fbSP_TemperatureLow(
	xEnable:= TRUE,		//rTemperature > 0,			//Temperature can drop below 0C
	rInput:= rTemperature, 
	rSwitchPoint:= rThresholdTemperatureLow_int, 
	rHysteresis:= 3, 
	xInvert:= TRUE, 
	xOut=> );
fbEI_TemperatureLow.sInstanceName := sInstanceName;
fbEI_TemperatureLow.sErrorInfo := TO_STRING(_Domoticz_RoundDecimals(rTemperature,1));
fbEI_TemperatureLow.sErrorInfo := CONCAT(fbEI_TemperatureLow.sErrorInfo, ' C');
fbEI_TemperatureLow(
	scConnector:= scConnector,
	xError:= fbSP_TemperatureLow.xOut
			AND rThresholdTemperatureLow_int > 0
			AND uiIdentifier_TempHumBaro > 0,
	eErrorID:= Domoticz_eErrors.Tasmota_TemperatureLow
);

//********************************************HUMIDITY
fbSP_HumidityHigh(	
	xEnable:= rHumidity > 0,								//If humidity not used (Temp or TempBaro)
	rInput:= rHumidity, 
	rSwitchPoint:= rThresholdHumidityHigh_int, 
	rHysteresis:= 10, 
	xInvert:= FALSE, 
	xOut=> );
fbEI_HumidityHigh.sInstanceName := sInstanceName;
fbEI_HumidityHigh.sErrorInfo := TO_STRING(TO_INT(_Domoticz_RoundDecimals(rHumidity,0)));
fbEI_HumidityHigh.sErrorInfo := CONCAT(fbEI_HumidityHigh.sErrorInfo, ' %');
fbEI_HumidityHigh(
	scConnector:= scConnector,
	xError:= fbSP_HumidityHigh.xOut 
			AND rThresholdHumidityHigh_int > 0
			AND uiIdentifier_TempHumBaro > 0,
	eErrorID:= Domoticz_eErrors.Tasmota_HumidityHigh
);

fbSP_HumidityLow(
	xEnable:= rHumidity > 0,								//If humidity not used (Temp or TempBaro)
	rInput:= rHumidity, 
	rSwitchPoint:= rThresholdHumidityLow_int, 
	rHysteresis:= 10, 
	xInvert:= TRUE, 
	xOut=> );
fbEI_HumidityLow.sInstanceName := sInstanceName;
fbEI_HumidityLow.sErrorInfo := TO_STRING(TO_INT(_Domoticz_RoundDecimals(rHumidity,0)));
fbEI_HumidityLow.sErrorInfo := CONCAT(fbEI_HumidityLow.sErrorInfo, ' %');
fbEI_HumidityLow(
	scConnector:= scConnector,
	xError:= fbSP_HumidityLow.xOut 							
			AND rThresholdHumidityLow_int > 0
			AND uiIdentifier_TempHumBaro > 0,
	eErrorID:= Domoticz_eErrors.Tasmota_HumidityLow
);

//********************************************CARBON DIOXIDE
fbSP_CarbonDioxideHigh(
	xEnable:= rCarbonDioxide > 0,
	rInput:= rCarbonDioxide, 
	rSwitchPoint:= rThresholdCarbonDioxideHigh_int, 
	rHysteresis:= 250, 
	xInvert:= FALSE, 
	xOut=> );
fbEI_CarbonDioxideHigh.sInstanceName := sInstanceName;
fbEI_CarbonDioxideHigh.sErrorInfo := TO_STRING(TO_INT(_Domoticz_RoundDecimals(rCarbonDioxide,0)));
fbEI_CarbonDioxideHigh.sErrorInfo := CONCAT(fbEI_CarbonDioxideHigh.sErrorInfo, ' ppm');
fbEI_CarbonDioxideHigh(
	scConnector:= scConnector,
	xError:= fbSP_CarbonDioxideHigh.xOut 
			AND rThresholdCarbonDioxideHigh_int > 0
			AND uiIdentifier_CarbonDioxide > 0,
	eErrorID:= Domoticz_eErrors.Tasmota_CarbondioxideHigh
);

fbSP_CarbonDioxideCritical(
	xEnable:= rCarbonDioxide > 0,
	rInput:= rCarbonDioxide, 
	rSwitchPoint:= rThresholdCarbonDioxideCritical_int, 
	rHysteresis:= 250, 
	xInvert:= FALSE, 
	xOut=> );
fbEI_CarbonDioxideCritical.sInstanceName := sInstanceName;
fbEI_CarbonDioxideCritical.sErrorInfo := TO_STRING(TO_INT(_Domoticz_RoundDecimals(rCarbonDioxide,0)));
fbEI_CarbonDioxideCritical.sErrorInfo := CONCAT(fbEI_CarbonDioxideCritical.sErrorInfo, ' ppm');
fbEI_CarbonDioxideCritical(
	scConnector:= scConnector,
	xError:= fbSP_CarbonDioxideCritical.xOut 
			AND rThresholdCarbonDioxideCritical_int > 0
			AND uiIdentifier_CarbonDioxide > 0,
	eErrorID:= Domoticz_eErrors.Tasmota_CarbonDioxideCritical
);

//********************************************PARTICLES
fbSP_1umHigh(
	xEnable:= rParticles_1um > 0,
	rInput:= rParticles_1um, 
	rSwitchPoint:= rThresholdParticlesHigh_1um_int, 
	rHysteresis:= 10, 
	xInvert:= FALSE, 
	xOut=> );
fbEI_1umHigh.sInstanceName := sInstanceName;
fbEI_1umHigh.sErrorInfo := TO_STRING(_Domoticz_RoundDecimals(rParticles_1um,1));
fbEI_1umHigh.sErrorInfo := CONCAT(fbEI_1umHigh.sErrorInfo, ' ug/m3');
fbEI_1umHigh(
	scConnector:= scConnector,
	xError:= fbSP_1umHigh.xOut
			AND rThresholdParticlesHigh_1um_int > 0
			AND uiIdentifier_1um > 0,
	eErrorID:= Domoticz_eErrors.Tasmota_ParticlesHigh_1um
);

fbSP_2_5umHigh(
	xEnable:= rParticles_2_5um > 0,
	rInput:= rParticles_2_5um, 
	rSwitchPoint:= rThresholdParticlesHigh_2_5um_int, 
	rHysteresis:= 10, 
	xInvert:= FALSE, 
	xOut=> );
fbEI_2_5umHigh.sInstanceName := sInstanceName;
fbEI_2_5umHigh.sErrorInfo := TO_STRING(_Domoticz_RoundDecimals(rParticles_2_5um,1));
fbEI_2_5umHigh.sErrorInfo := CONCAT(fbEI_2_5umHigh.sErrorInfo, ' ug/m3');
fbEI_2_5umHigh(
	scConnector:= scConnector,
	xError:= fbSP_2_5umHigh.xOut 
			AND rThresholdParticlesHigh_2_5um_int > 0
			AND uiIdentifier_2_5um > 0,
	eErrorID:= Domoticz_eErrors.Tasmota_ParticlesHigh_2_5um
);

fbSP_10umHigh(	
	xEnable:= rParticles_10um > 0,
	rInput:= rParticles_10um,
	rSwitchPoint:= rThresholdParticlesHigh_10um_int, 
	rHysteresis:= 10, 
	xInvert:= FALSE, 
	xOut=> );
fbEI_10umHigh.sInstanceName := sInstanceName;
fbEI_10umHigh.sErrorInfo := TO_STRING(_Domoticz_RoundDecimals(rParticles_10um,1));
fbEI_10umHigh.sErrorInfo := CONCAT(fbEI_10umHigh.sErrorInfo, ' ug/m3');
fbEI_10umHigh(
	scConnector:= scConnector,
	xError:= fbSP_10umHigh.xOut 
			AND rThresholdParticlesHigh_10um_int > 0
			AND uiIdentifier_10um > 0,
	eErrorID:= Domoticz_eErrors.Tasmota_ParticlesHigh_10um
);
END_ACTION

{attribute 'monitoring' := 'call'} PROPERTY rThresholdCurrentHigh :REAL
SET
rThresholdCurrentHigh_int := rThresholdCurrentHigh;
END_SET
GET
rThresholdCurrentHigh := rThresholdCurrentHigh_int;
END_GET
END_PROPERTY

{attribute 'monitoring' := 'call'} PROPERTY rThresholdCurrentMax :REAL
SET
rThresholdCurrentMax_int := rThresholdCurrentMax;
END_SET
GET
rThresholdCurrentMax := rThresholdCurrentMax_int;
END_GET
END_PROPERTY

{attribute 'monitoring' := 'call'} PROPERTY rThresholdPowerUsageHigh :REAL
SET
rThresholdPowerUsageHigh_int := rThresholdPowerUsageHigh;
END_SET
GET
rThresholdPowerUsageHigh := rThresholdPowerUsageHigh_int;
END_GET
END_PROPERTY

{attribute 'monitoring' := 'call'} PROPERTY rThresholdPowerUsageToday :REAL
SET
rThresholdPowerUsageToday_int := rThresholdPowerUsageToday;
END_SET
GET
rThresholdPowerUsageToday := rThresholdPowerUsageToday_int;
END_GET
END_PROPERTY

{attribute 'monitoring' := 'call'} PROPERTY rThresholdTemperatureHigh :REAL
SET
rThresholdTemperatureHigh_int := rThresholdTemperatureHigh;
END_SET
GET
rThresholdTemperatureHigh := rThresholdTemperatureHigh_int;
END_GET
END_PROPERTY

{attribute 'monitoring' := 'call'} PROPERTY rThresholdTemperatureLow :REAL
SET
rThresholdTemperatureLow_int := rThresholdTemperatureLow;
END_SET
GET
rThresholdTemperatureLow := rThresholdTemperatureLow_int;
END_GET
END_PROPERTY

{attribute 'monitoring' := 'call'} PROPERTY rThresholdHumidityHigh :REAL
SET
rThresholdHumidityHigh_int := rThresholdHumidityHigh;
END_SET
GET
rThresholdHumidityHigh := rThresholdHumidityHigh_int;
END_GET
END_PROPERTY

{attribute 'monitoring' := 'call'} PROPERTY rThresholdHumidityLow :REAL
SET
rThresholdHumidityLow_int := rThresholdHumidityLow;
END_SET
GET
rThresholdHumidityLow := rThresholdHumidityLow_int;
END_GET
END_PROPERTY

{attribute 'monitoring' := 'call'} PROPERTY rThresholdCarbonDioxideHigh :REAL
SET
rThresholdCarbonDioxideHigh_int := rThresholdCarbonDioxideHigh;
END_SET
GET
rThresholdCarbonDioxideHigh := rThresholdCarbonDioxideHigh_int;
END_GET
END_PROPERTY

{attribute 'monitoring' := 'call'} PROPERTY rThresholdCarbonDioxideCritical :REAL
SET
rThresholdCarbonDioxideCritical_int := rThresholdCarbonDioxideCritical;
END_SET
GET
rThresholdCarbonDioxideCritical := rThresholdCarbonDioxideCritical_int;
END_GET
END_PROPERTY

{attribute 'monitoring' := 'call'} PROPERTY rThresholdParticlesHigh_1um :REAL
SET
rThresholdParticlesHigh_1um_int := rThresholdParticlesHigh_1um;
END_SET
GET
rThresholdParticlesHigh_1um := rThresholdParticlesHigh_1um_int;
END_GET
END_PROPERTY

{attribute 'monitoring' := 'call'} PROPERTY rThresholdParticlesHigh_2_5um :REAL
SET
rThresholdParticlesHigh_2_5um_int := rThresholdParticlesHigh_2_5um;
END_SET
GET
rThresholdParticlesHigh_2_5um := rThresholdParticlesHigh_2_5um_int;
END_GET
END_PROPERTY

{attribute 'monitoring' := 'call'} PROPERTY rThresholdParticlesHigh_10um :REAL
SET
rThresholdParticlesHigh_10um_int := rThresholdParticlesHigh_10um;
END_SET
GET
rThresholdParticlesHigh_10um := rThresholdParticlesHigh_10um_int;
END_GET
END_PROPERTY

PROPERTY rThresholdVoltage : REAL
SET
rThresholdVoltage_int := rThresholdVoltage;
END_SET
GET
rThresholdVoltage := rThresholdVoltage_int;
END_GET
END_PROPERTY

END_FUNCTION_BLOCK

// Function Blocks/Hardware/Devices/Domoticz_GoogleDevices
{attribute 'conditionalshow_all_locals'}
FUNCTION_BLOCK Domoticz_GoogleDevices EXTENDS _Domoticz_Connector_InOut	//Don't use xForceValues for everything because it will also force byMediaControl_Set
VAR_INPUT
	uiIdentifier_Status			:UINT;	//Device Status
	uiIdentifier_Source			:UINT;	//Source of active footage
	uiIdentifier_Volume			:UINT;	//Device Volume
	byVolume_Set				:BYTE;	//Volume (0-100)
	uiIdentifier_MediaControl	:UINT;	//Process Usage
	byMediaControl_Set			:BYTE;	//Play process (0-100)
	xMediaControl_Set			:BOOL;	//Play media
END_VAR
VAR_OUTPUT
	sStatus						:STRING(Domoticz_Constants.uiMaxSValuesize);
	bySource					:BYTE;	//See domoticz settings! Default:0=off, 10=Spotify, 20=Netflix, 30=Youtube, 40=Other
	byVolume_Act				:BYTE;
	byMediaControl_Act			:BYTE;
	xMediaControl_Act			:BOOL;
END_VAR
VAR
	afb_ObjectString_Out		:ARRAY[1..1] OF _Domoticz_ObjectString_Out;
	afb_ObjectInt_Out			:ARRAY[1..1] OF _Domoticz_ObjectInt_Out;
	afb_ObjectInt_InOut			:ARRAY[1..2] OF _Domoticz_ObjectInt_InOut;
	afb_ObjectBool_InOut		:ARRAY[1..1] OF _Domoticz_ObjectBool_InOut;
END_VAR

IF __ISVALIDREF(scConnector) THEN
	Main();
END_IF

ACTION Main:
{attribute 'conditionalshow'}
//Call parent function
SUPER^.Main();

//Call all 
afb_ObjectString_Out[1].tDataTimeOut := T#24H;
afb_ObjectString_Out[1](scConnector := scConnector,		uiIdentifier := uiIdentifier_Status,		rxUpdateInterlock := rxUpdateInterlock_int,			sValueAct => sStatus);

afb_ObjectInt_Out[1].tDataTimeOut := T#24H;
afb_ObjectInt_Out[1](	scConnector := scConnector,		uiIdentifier := uiIdentifier_Source,		rxUpdateInterlock := rxUpdateInterlock_int);

afb_ObjectInt_InOut[1].tDataTimeOut := T#24H;
afb_ObjectInt_InOut[1].iValueSetLimitLow := -1;
afb_ObjectInt_InOut[1].iValueSetLimitHigh := 101;
afb_ObjectInt_InOut[1].eCommandType := _Domoticz_eCommandType.SetBrightness;
afb_ObjectInt_InOut[1](	scConnector := scConnector, 	uiIdentifier := uiIdentifier_Volume,		rxUpdateInterlock := rxUpdateInterlock_int,			iValueSet := byVolume_Set);

afb_ObjectInt_InOut[2].tDataTimeOut := T#24H;
afb_ObjectInt_InOut[2].iValueSetLimitLow := -1;
afb_ObjectInt_InOut[2].iValueSetLimitHigh := 101;
afb_ObjectInt_InOut[2].eCommandType := _Domoticz_eCommandType.SetBrightness;
afb_ObjectInt_InOut[2](	scConnector := scConnector, 	uiIdentifier := uiIdentifier_MediaControl,	rxUpdateInterlock := rxUpdateInterlock_int,			iValueSet := byMediaControl_Set);

afb_ObjectBool_InOut[1].tDataTimeOut := T#24H;      
afb_ObjectBool_InOut[1].eCommandType := _Domoticz_eCommandType.SwitchLight;                                                 
afb_ObjectBool_InOut[1](scConnector := scConnector,		uiIdentifier := uiIdentifier_MediaControl,	rxUpdateInterlock := rxUpdateInterlock_int,			xValueSet := xMediaControl_Set,		xValueAct => xMediaControl_Act);
						
//Output
bySource 			:= TO_BYTE(afb_ObjectInt_Out[1].iValueAct);
byVolume_Act 		:= TO_BYTE(afb_ObjectInt_InOut[1].iValueAct);
byMediaControl_Act 	:= TO_BYTE(afb_ObjectInt_InOut[2].iValueAct);
 
//Force update of volume
IF xForceSetValues AND byVolume_Set <> byVolume_Act THEN
	afb_ObjectInt_InOut[1].ForceSet(tForceSetValues_int);
END_IF

//Force update of media control
IF xForceSetValues AND byMediaControl_Set <> byMediaControl_Act THEN
	afb_ObjectInt_InOut[2].ForceSet(tForceSetValues_int);
END_IF

//Force update of media control
IF xForceSetValues AND xMediaControl_Set <> xMediaControl_Act THEN
	afb_ObjectBool_InOut[1].ForceSet(tForceSetValues_int);
END_IF
										   
//Errors
fbEI_DataTimeOut.sInstanceName := sInstanceName;
fbEI_DataTimeOut.tErrorDelay := T#500MS;	//Give objects time to be overruled by other updates
fbEI_DataTimeOut(
	scConnector:= scConnector,
	xError:= xDataTimeOut_int
			AND (afb_ObjectString_Out[1].xDataTimedOut
			OR afb_ObjectInt_Out[1].xDataTimedOut
			OR afb_ObjectInt_InOut[1].xDataTimedOut
			OR afb_ObjectInt_InOut[2].xDataTimedOut
			OR afb_ObjectBool_InOut[1].xDataTimedOut),
	eErrorID:= Domoticz_eErrors.ObjectDataTimeOut
);
END_ACTION

END_FUNCTION_BLOCK

// Function Blocks/Hardware/Custom/Domoticz_CustomString
{attribute 'conditionalshow_all_locals'}
FUNCTION_BLOCK Domoticz_CustomString EXTENDS _Domoticz_Connector_InOut_Extended
VAR_INPUT
	uiIdentifier				:UINT;	//Device to control
	sValueSet					:STRING(Domoticz_Constants.uiMaxSValuesize);
END_VAR
VAR_OUTPUT
	sValueAct					:STRING(Domoticz_Constants.uiMaxSValuesize);
END_VAR
VAR
	afb_ObjectString_InOut		:ARRAY[1..1] OF _Domoticz_ObjectString_InOut;
END_VAR

IF __ISVALIDREF(scConnector) THEN
	Main();
END_IF

ACTION Main:
{attribute 'conditionalshow'}
//Call parent function
SUPER^.Main();

//Call all functions
afb_ObjectString_InOut[1].tDataTimeOut := tDataTimeOut_int;
afb_ObjectString_InOut[1](scConnector := scConnector, 	uiIdentifier := uiIdentifier,	sValueSet := sValueSet, 	sValueAct => sValueAct);

//Force status if enabled
IF xForceSetValues AND sValueSet <> sValueAct THEN
	afb_ObjectString_InOut[1].ForceSet(tForceSetValues_int);
END_IF

//Errors
fbEI_DataTimeOut.sInstanceName := sInstanceName;
fbEI_DataTimeOut.tErrorDelay := T#500MS;	//Give objects TIME TO be overruled BY other updates
fbEI_DataTimeOut(
	scConnector:= scConnector,
	xError:= xDataTimeOut_int
			AND (afb_ObjectString_InOut[1].xDataTimedOut),
	eErrorID:= Domoticz_eErrors.ObjectDataTimeOut
);
END_ACTION

END_FUNCTION_BLOCK

// Function Blocks/Hardware/Climate/Energy/Domoticz_UsageMeter
{attribute 'conditionalshow_all_locals'}
FUNCTION_BLOCK Domoticz_UsageMeter EXTENDS _Domoticz_Connector_Out
VAR_INPUT
	uiIdentifier_Usage			:UINT;			//Usage (cumulative)
	xPulse						:BOOL;			//Measure pulse
	rUnitsPerPulse				:REAL := 1000;	//Units per pulse
	rUnitsBeforeUpdate			:REAL := 1000;	//Amount of units to reach before sending update
	tTimeOutPulse				:TIME := T#5M;	//Time to pass without pulses to sens stored values
END_VAR                          
VAR_OUTPUT                       
	rUsageToday					:REAL;
	rUsageCumulative			:REAL;
END_VAR                          
VAR	                             
	afb_ObjectArrayReal_InOut	:ARRAY[1..1] OF _Domoticz_ObjectArrayReal_InOut;
	xPulse_old					:BOOL;
	TON_TimeOutPulse			:TON;
	                             
	rThresholdUsageToday_int	:REAL := 500;
	fbEI_UsageToday				:Domoticz_ErrorInterface;
	
	sUnit_int					:STRING := 'm3';
END_VAR                          
VAR PERSISTENT RETAIN                 
	rPulsesCounted				:REAL;
END_VAR

IF __ISVALIDREF(scConnector) THEN
	Main();
END_IF

ACTION Main:
{attribute 'conditionalshow'}
//Call parent function
SUPER^.Main();

//Add usage on pulse
IF xPulse AND NOT xPulse_old THEN
	xPulse_old := TRUE;
	//Add pulses if limit not reached, set data to zero
	IF ((rPulsesCounted+1)*rUnitsPerPulse) < rUnitsBeforeUpdate THEN
		rPulsesCounted := rPulsesCounted + 1;
		afb_ObjectArrayReal_InOut[1].arValueSet[Domoticz_eSValues_Usage.Usage] := 0;
	//Limit reached, send data and reset counter
	ELSIF ((rPulsesCounted+1)*rUnitsPerPulse) >= rUnitsBeforeUpdate THEN
		afb_ObjectArrayReal_InOut[1].arValueSet[Domoticz_eSValues_Usage.Usage] := rUnitsBeforeUpdate;
		rPulsesCounted := 0;
	END_IF
//Reset flank
ELSIF NOT xPulse THEN
	xPulse_old := FALSE;
END_IF
	
//Send usage after timeout to prevent values buildup
IF TON_TimeOutPulse.Q THEN
	afb_ObjectArrayReal_InOut[1].arValueSet[Domoticz_eSValues_Usage.Usage] := rPulsesCounted*rUnitsPerPulse;
	rPulsesCounted := 0;
END_IF

//Call all functions
afb_ObjectArrayReal_InOut[1].tDataTimeOut := T#15M;
afb_ObjectArrayReal_InOut[1].eDataSource := _Domoticz_eDataSource.HTTP;
afb_ObjectArrayReal_InOut[1](scConnector := scConnector, 	uiIdentifier := uiIdentifier_Usage);

//Call timer
TON_TimeOutPulse(IN:= NOT xPulse, PT:= tTimeOutPulse);

//Outputs
rUsageToday := afb_ObjectArrayReal_InOut[1].arValueAct[Domoticz_eSValues_Usage.UsageToday];
rUsageCumulative := afb_ObjectArrayReal_InOut[1].arValueAct[Domoticz_eSValues_Usage.UsageCumulative];

//Errors
//********************************************DATA
fbEI_DataTimeOut.sInstanceName := sInstanceName;
fbEI_DataTimeOut.tErrorDelay := T#500MS;	//Give objects TIME TO be overruled BY other updates
fbEI_DataTimeOut(
	scConnector:= scConnector,
	xError:= xDataTimeOut_int
			AND (afb_ObjectArrayReal_InOut[1].xDataTimedOut),
	eErrorID:= Domoticz_eErrors.ObjectDataTimeOut
);

//********************************************USAGE TODAY
fbEI_UsageToday.sInstanceName := sInstanceName;
fbEI_UsageToday.sErrorInfo := TO_STRING(_Domoticz_RoundDecimals(rUsageToday,2));
fbEI_UsageToday.sErrorInfo := CONCAT(fbEI_UsageToday.sErrorInfo, ' ');
fbEI_UsageToday.sErrorInfo := CONCAT(fbEI_UsageToday.sErrorInfo, sUnit_int);
fbEI_UsageToday(
	scConnector:= scConnector,
	xError:= (rUsageToday > rThresholdUsageToday_int) 
			AND rThresholdUsageToday_int > 0
			AND uiIdentifier_Usage > 0,
	eErrorID:= Domoticz_eErrors.UsageMeter_UsageToday
);
END_ACTION

{attribute 'monitoring' := 'call'} PROPERTY rThresholdUsageToday :REAL
SET
rThresholdUsageToday_int := rThresholdUsageToday;
END_SET
GET
rThresholdUsageToday := rThresholdUsageToday_int;
END_GET
END_PROPERTY

PROPERTY sUnit : STRING
SET
sUnit_int := sUnit;
END_SET
GET
sUnit := sUnit_int;
END_GET
END_PROPERTY

END_FUNCTION_BLOCK

// Function Blocks/Hardware/Devices/Domoticz_Life360
{attribute 'conditionalshow_all_locals'}
//Function block to update sentire values in domoticz
FUNCTION_BLOCK Domoticz_Life360 EXTENDS _Domoticz_Connector_Out
VAR_INPUT
	uiIdentifier_Presence				:UINT;	//Presence at home
	uiIdentifier_Location				:UINT;	//Current location (text)
	uiIdentifier_Battery				:UINT;	//Device battery (%)
	uiIdentifier_Distance				:UINT;	//Distance to home
END_VAR
VAR_OUTPUT
	xPresence							:BOOL;
	sLocation							:STRING;
	rBattery							:REAL;
	sDistance							:STRING;
END_VAR
VAR
	afb_ObjectReal_Out					:ARRAY[1..1] OF _Domoticz_ObjectReal_Out;
	afb_ObjectString_Out				:ARRAY[1..2] OF _Domoticz_ObjectString_Out;		
	afb_ObjectBool_Out					:ARRAY[1..1] OF _Domoticz_ObjectBool_Out;
	
	xArrivedHome_int					:BOOL := TRUE;
	fbEI_ArrivedHome					:Domoticz_ErrorInterface;
	
	xLeftHome_int						:BOOL := TRUE;
	fbEI_LeftHome						:Domoticz_ErrorInterface;
	
END_VAR

IF __ISVALIDREF(scConnector) THEN
	Main();
END_IF

ACTION Main:
{attribute 'conditionalshow'}
//Call parent function
SUPER^.Main();

//Call all functions
//Data timeout assume normal workweek - excluding weekends
afb_ObjectReal_Out[1].tDataTimeOut := T#3D;
afb_ObjectReal_Out[1](scConnector := scConnector, 	uiIdentifier := uiIdentifier_Battery,		rxUpdateInterlock := rxUpdateInterlock_int,			rValueAct => rBattery);
                                                                                            	                                                	
afb_ObjectBool_Out[1].tDataTimeOut := T#3D;                                                 	                                                	
afb_ObjectBool_Out[1](scConnector:= scConnector, 	uiIdentifier:= uiIdentifier_Presence,		rxUpdateInterlock := rxUpdateInterlock_int,			xValueAct => xPresence);
                                                                                            	                                                	
afb_ObjectString_Out[1].tDataTimeOut := T#3D;                                               	                                                	
afb_ObjectString_Out[1](scConnector := scConnector,	uiIdentifier := uiIdentifier_Location,		rxUpdateInterlock := rxUpdateInterlock_int,			sValueAct => sLocation);
                                                                                            	                                                	
afb_ObjectString_Out[2].tDataTimeOut := T#3D;                                               	                                                	
afb_ObjectString_Out[2](scConnector := scConnector,	uiIdentifier := uiIdentifier_Distance, 		rxUpdateInterlock := rxUpdateInterlock_int,			sValueAct => sDistance);

//Errors
fbEI_DataTimeOut.sInstanceName := sInstanceName;
fbEI_DataTimeOut.tErrorDelay := T#500MS;	//Give objects TIME TO be overruled BY other updates
fbEI_DataTimeOut(
	scConnector:= scConnector,
	xError:= xDataTimeOut_int
			AND (afb_ObjectReal_Out[1].xDataTimedOut
			OR afb_ObjectBool_Out[1].xDataTimedOut
			OR afb_ObjectString_Out[1].xDataTimedOut
			OR afb_ObjectString_Out[2].xDataTimedOut),
	eErrorID:= Domoticz_eErrors.ObjectDataTimeOut
);

fbEI_ArrivedHome.sInstanceName := sInstanceName;
fbEI_ArrivedHome(
	scConnector:= scConnector, 
	xError:= xPresence
			AND xArrivedHome_int, 
	eErrorID:= Domoticz_eErrors.Life360_ArrivedHome
);

fbEI_LeftHome.sInstanceName := sInstanceName;
fbEI_LeftHome(
	scConnector:= scConnector, 
	xError:= NOT xPresence
			AND xleftHome_int, 
	eErrorID:= Domoticz_eErrors.Life360_LeftHome
);
END_ACTION

PROPERTY xArrivedHome :BOOL
SET
xArrivedHome_int := xArrivedHome;
END_SET
GET
xArrivedHome := xArrivedHome_int;
END_GET
END_PROPERTY

PROPERTY xLeftHome :BOOL
SET
xLeftHome_int := xLeftHome;
END_SET
GET
xLeftHome := xLeftHome_int;
END_GET
END_PROPERTY

END_FUNCTION_BLOCK

// Function Blocks/Hardware/Devices/Domoticz_HueSensor
{attribute 'conditionalshow_all_locals'}
//Function block to update sentire values in domoticz
FUNCTION_BLOCK Domoticz_HueSensor EXTENDS _Domoticz_Connector_Out
VAR_INPUT
	uiIdentifier_Temperature			:UINT;	//Temperature (C)
	uiIdentifier_Light					:UINT;	//Light level (lux)
	uiIdentifier_Ambient				:UINT;	//Ambient light level
	uiIdentifier_PIR					:UINT;	//PIR
END_VAR
VAR_OUTPUT
	rTemperature						:REAL;
	rLightIntensity						:REAL;
	xAmbient							:BOOL;
	xPIR								:BOOL;
END_VAR
VAR
	afb_ObjectReal_Out					:ARRAY[1..2] OF _Domoticz_ObjectReal_Out;
	afb_ObjectBool_Out					:ARRAY[1..2] OF _Domoticz_ObjectBool_Out;
END_VAR

IF __ISVALIDREF(scConnector) THEN
	Main();
END_IF

ACTION Main:
{attribute 'conditionalshow'}
//Call parent function
SUPER^.Main();

//Call all functions
//Data timeout Light/temp depend on amount of changes, assume 4h. Ambient switch at least twice a day
afb_ObjectReal_Out[1].tDataTimeOut := T#4H;
afb_ObjectReal_Out[1](scConnector:= scConnector,	uiIdentifier:= uiIdentifier_Temperature,		rxUpdateInterlock := rxUpdateInterlock_int,			rValueAct=> rTemperature);

afb_ObjectReal_Out[2].tDataTimeOut := T#8H;
afb_ObjectReal_Out[2](scConnector:= scConnector,	uiIdentifier:= uiIdentifier_Light,				rxUpdateInterlock := rxUpdateInterlock_int,			rValueAct=> rLightIntensity);

afb_ObjectBool_Out[1].tDataTimeOut := T#24H;	//Not guarded PIR
afb_ObjectBool_Out[1](scConnector:= scConnector, 	uiIdentifier:= uiIdentifier_PIR,				rxUpdateInterlock := rxUpdateInterlock_int,			xValueAct=> xPIR);

afb_ObjectBool_Out[2].tDataTimeOut := T#24H;
afb_ObjectBool_Out[2](scConnector:= scConnector, 	uiIdentifier:= uiIdentifier_Ambient,			rxUpdateInterlock := rxUpdateInterlock_int,			xValueAct=> xAmbient);									
										   
//Errors
fbEI_DataTimeOut.sInstanceName := sInstanceName;
fbEI_DataTimeOut.tErrorDelay := T#500MS;	//Give objects TIME TO be overruled BY other updates
fbEI_DataTimeOut(
	scConnector:= scConnector,
	xError:= xDataTimeOut_int
			AND (afb_ObjectReal_Out[1].xDataTimedOut
			OR afb_ObjectReal_Out[2].xDataTimedOut
			OR afb_ObjectBool_Out[1].xDataTimedOut
			OR afb_ObjectBool_Out[2].xDataTimedOut),
	eErrorID:= Domoticz_eErrors.ObjectDataTimeOut
);
END_ACTION

END_FUNCTION_BLOCK

// Function Blocks/Hardware/Devices/Domoticz_HuePlug
{attribute 'conditionalshow_all_locals'}
FUNCTION_BLOCK Domoticz_HuePlug EXTENDS _Domoticz_Connector_InOut
VAR_INPUT
	uiIdentifier				:UINT;	//Device to control
	xEnable						:BOOL;
END_VAR
VAR_OUTPUT
	xEnabled					:BOOL;
END_VAR
VAR
	afb_ObjectBool_InOut		:ARRAY[1..1] OF _Domoticz_ObjectBool_InOut;
END_VAR

IF __ISVALIDREF(scConnector) THEN
	Main();
END_IF

ACTION Main:
{attribute 'conditionalshow'}
//Call parent function
SUPER^.Main();

//Call all functions
afb_ObjectBool_InOut[1].tDataTimeOut := T#24H;
afb_ObjectBool_InOut[1].eCommandType := _Domoticz_eCommandType.SwitchLight;
afb_ObjectBool_InOut[1](scConnector := scConnector, 	uiIdentifier := uiIdentifier, 	xValueSet := xEnable, 	xValueAct => xEnabled);

//Force status if enabled
IF xForceSetValues AND xEnable <> xEnabled THEN
	afb_ObjectBool_InOut[1].ForceSet(tForceSetValues_int);
END_IF

//Errors
fbEI_DataTimeOut.sInstanceName := sInstanceName;
fbEI_DataTimeOut.tErrorDelay := T#500MS;	//Give objects TIME TO be overruled BY other updates
fbEI_DataTimeOut(
	scConnector:= scConnector,
	xError:= xDataTimeOut_int
			AND (afb_ObjectBool_InOut[1].xDataTimedOut),
	eErrorID:= Domoticz_eErrors.ObjectDataTimeOut
);
END_ACTION

END_FUNCTION_BLOCK

// Function Blocks/Hardware/Climate/Energy/Domoticz_P1Meter
{attribute 'conditionalshow_all_locals'}
FUNCTION_BLOCK Domoticz_P1Meter EXTENDS _Domoticz_Connector_Out
VAR_INPUT
	uiIdentifier_Voltage		:UINT;				//Usage
	uiIdentifier_Power			:UINT;				//Usage
	uiIdentifier_Gas			:UINT;				//Usage
	tUpdateRate					:TIME := T#60M;		//Used for data timeout
END_VAR                          
VAR_OUTPUT                       
	rVoltage					:REAL;
	rPowerUsageActual			:REAL;
	rPowerUsageToday			:REAL;
	rPowerUsageCumulative		:REAL;
	rPowerReturnActual			:REAL;
	rPowerReturnToday			:REAL;
	rPowerReturnCumulative		:REAL;
	rGasUsageToday				:REAL;
	rGasUsageCumulative			:REAL;
END_VAR                          
VAR	                             
	afb_ObjectReal_Out			:ARRAY[1..1] OF _Domoticz_ObjectReal_Out;
	afb_ObjectArrayReal_Out		:ARRAY[1..2] OF _Domoticz_ObjectArrayReal_Out;
	                             
	rThresholdVoltage_int		:REAL := 200;
	fbEI_PowerFailure			:Domoticz_ErrorInterface;
	                             
	rThresholdPowerUsageToday_int:REAL := 10.0; //kWh
	fbEI_PowerUsageToday		:Domoticz_ErrorInterface;
	                             
	rThresholdPowerUsageHigh_int:REAL := 3000;	//W
	fbSP_PowerUsageHigh			:_Domoticz_SwitchPoint;
	fbEI_PowerUsageHigh			:Domoticz_ErrorInterface;
	                             
	rThresholdGasUsageToday_int	:REAL := 5.0;	//m3
	fbEI_GasUsageToday			:Domoticz_ErrorInterface;
END_VAR

IF __ISVALIDREF(scConnector) THEN
	Main();
END_IF

ACTION Main:
{attribute 'conditionalshow'}
//Call parent function
SUPER^.Main();

//Call all functions
afb_ObjectReal_Out[1].tDataTimeOut := TO_TIME(TO_UDINT(tUpdateRate)*2);
afb_ObjectReal_Out[1](	scConnector := scConnector, 	uiIdentifier := uiIdentifier_Voltage, 		rxUpdateInterlock := rxUpdateInterlock_int,			rValueAct => rVoltage);

afb_ObjectArrayReal_Out[1].tDataTimeOut := TO_TIME(TO_UDINT(tUpdateRate)*2);
afb_ObjectArrayReal_Out[1](	scConnector := scConnector, uiIdentifier := uiIdentifier_Gas,			rxUpdateInterlock := rxUpdateInterlock_int);

afb_ObjectArrayReal_Out[2].tDataTimeOut := TO_TIME(TO_UDINT(tUpdateRate)*2);
afb_ObjectArrayReal_Out[2](scConnector := scConnector, 	uiIdentifier := uiIdentifier_Power,			rxUpdateInterlock := rxUpdateInterlock_int);

//Outputs
rGasUsageCumulative		:= afb_ObjectArrayReal_Out[1].arValueAct[Domoticz_eSValues_P1.Usage1Cumulative] + afb_ObjectArrayReal_Out[1].arValueAct[Domoticz_eSValues_P1.Usage2Cumulative];
rGasUsageToday			:= afb_ObjectArrayReal_Out[1].arValueAct[Domoticz_eSValues_P1.UsageToday];

rPowerUsageActual 		:= afb_ObjectArrayReal_Out[2].arValueAct[Domoticz_eSValues_P1.UsageActual];
rPowerReturnActual 		:= afb_ObjectArrayReal_Out[2].arValueAct[Domoticz_eSValues_P1.ReturnActual];
rPowerUsageCumulative 	:= afb_ObjectArrayReal_Out[2].arValueAct[Domoticz_eSValues_P1.Usage1Cumulative] + afb_ObjectArrayReal_Out[2].arValueAct[Domoticz_eSValues_P1.Usage2Cumulative];
rPowerReturnCumulative	:= afb_ObjectArrayReal_Out[2].arValueAct[Domoticz_eSValues_P1.Return1Cumulative] + afb_ObjectArrayReal_Out[2].arValueAct[Domoticz_eSValues_P1.Return2Cumulative];	
rPowerUsageToday 		:= afb_ObjectArrayReal_Out[2].arValueAct[Domoticz_eSValues_P1.UsageToday];
rPowerReturnToday 		:= afb_ObjectArrayReal_Out[2].arValueAct[Domoticz_eSValues_P1.ReturnToday];

//Errors
//********************************************DATA
fbEI_DataTimeOut.sInstanceName := sInstanceName;
fbEI_DataTimeOut.tErrorDelay := T#500MS;	//Give objects TIME TO be overruled BY other updates
fbEI_DataTimeOut(
	scConnector:= scConnector,
	xError:= xDataTimeOut_int
			AND (afb_ObjectReal_Out[1].xDataTimedOut
			OR afb_ObjectArrayReal_Out[1].xDataTimedOut
			OR afb_ObjectArrayReal_Out[2].xDataTimedOut),
	eErrorID:= Domoticz_eErrors.ObjectDataTimeOut
);

//********************************************POWER FAILURE
fbEI_PowerFailure.sInstanceName := sInstanceName;
fbEI_PowerFailure.sErrorInfo := TO_STRING(TO_INT(_Domoticz_RoundDecimals(rVoltage,0)));
fbEI_PowerFailure.sErrorInfo := CONCAT(fbEI_PowerFailure.sErrorInfo, ' V / ');
fbEI_PowerFailure.sErrorInfo := CONCAT(fbEI_PowerFailure.sErrorInfo, TO_STRING(TO_INT(_Domoticz_RoundDecimals(rPowerUsageActual,0))));
fbEI_PowerFailure.sErrorInfo := CONCAT(fbEI_PowerFailure.sErrorInfo, ' W');
fbEI_PowerFailure(
	scConnector:= scConnector,
	xError:= ((rVoltage < rThresholdVoltage_int) OR (rPowerUsageActual < 1)) 
			AND (uiIdentifier_Voltage > 0 OR  uiIdentifier_Power > 0),
	eErrorID:= Domoticz_eErrors.P1_PowerFailure
);

//********************************************USAGE TODAY
fbEI_PowerUsageToday.sInstanceName := sInstanceName;
fbEI_PowerUsageToday.sErrorInfo := TO_STRING(_Domoticz_RoundDecimals(rPowerUsageToday,2));
fbEI_PowerUsageToday.sErrorInfo := CONCAT(fbEI_PowerUsageToday.sErrorInfo, ' kWh');
fbEI_PowerUsageToday(
	scConnector:= scConnector,
	xError:= (rPowerUsageToday > rThresholdPowerUsageToday_int) 
			AND rThresholdPowerUsageToday_int > 0
			AND uiIdentifier_Power > 0,
	eErrorID:= Domoticz_eErrors.P1_PowerUsageToday
);

//********************************************USAGE
fbSP_PowerUsageHigh(
	xEnable:= rPowerUsageActual > 0,
	rInput:= rPowerUsageActual, 
	rSwitchPoint:= rThresholdPowerUsageHigh_int, 
	rHysteresis:= 500, 
	xInvert:= FALSE, 
	xOut=> );
fbEI_PowerUsageHigh.sInstanceName := sInstanceName;
fbEI_PowerUsageHigh.sErrorInfo := TO_STRING(TO_INT(_Domoticz_RoundDecimals(rPowerUsageActual,0)));
fbEI_PowerUsageHigh.sErrorInfo := CONCAT(fbEI_PowerUsageHigh.sErrorInfo, ' W');
fbEI_PowerUsageHigh(
	scConnector:= scConnector,
	xError:= fbSP_PowerUsageHigh.xOut
			AND rThresholdPowerUsageHigh_int > 0
			AND uiIdentifier_Power > 0,
	eErrorID:= Domoticz_eErrors.P1_PowerUsageHigh
);

//********************************************USAGE TODAY
fbEI_GasUsageToday.sInstanceName := sInstanceName;
fbEI_GasUsageToday.sErrorInfo := TO_STRING(_Domoticz_RoundDecimals(rGasUsageToday,2));
fbEI_GasUsageToday.sErrorInfo := CONCAT(fbEI_GasUsageToday.sErrorInfo, ' m3');
fbEI_GasUsageToday(
	scConnector:= scConnector,
	xError:= (rGasUsageToday > rThresholdGasUsageToday_int) 
			AND rThresholdGasUsageToday_int > 0
			AND uiIdentifier_Gas > 0,
	eErrorID:= Domoticz_eErrors.P1_GasUsageToday
);
END_ACTION

{attribute 'monitoring' := 'call'} PROPERTY rThresholdGasUsageToday :REAL
SET
rThresholdGasUsageToday_int := rThresholdGasUsageToday;
END_SET
GET
rThresholdGasUsageToday := rThresholdGasUsageToday_int;
END_GET
END_PROPERTY

{attribute 'monitoring' := 'call'} PROPERTY rThresholdPowerUsageHigh :REAL
SET
rThresholdPowerUsageHigh_int := rThresholdPowerUsageHigh;
END_SET
GET
rThresholdPowerUsageHigh := rThresholdPowerUsageHigh_int;
END_GET
END_PROPERTY

{attribute 'monitoring' := 'call'} PROPERTY rThresholdPowerUsageToday :REAL
SET
rThresholdPowerUsageToday_int := rThresholdPowerUsageToday;
END_SET
GET
rThresholdPowerUsageToday := rThresholdPowerUsageToday_int;
END_GET
END_PROPERTY

PROPERTY rThresholdVoltage : REAL
SET
rThresholdVoltage_int := rThresholdVoltage;
END_SET
GET
rThresholdVoltage := rThresholdVoltage_int;
END_GET
END_PROPERTY

END_FUNCTION_BLOCK

// Function Blocks/Hardware/Devices/Domoticz_HueSwitch
{attribute 'conditionalshow_all_locals'}
FUNCTION_BLOCK Domoticz_HueSwitch EXTENDS _Domoticz_Connector_Out
VAR_INPUT
	uiIdentifier				:UINT;	//Device to control
END_VAR
VAR_OUTPUT
	axButtons_Short				:ARRAY[1..4] OF BOOL;
	axButtons_Long				:ARRAY[1..4] OF BOOL;
END_VAR
VAR
	afb_ObjectInt_Out			:ARRAY[1..1] OF _Domoticz_ObjectInt_Out;
	wX							:WORD;
END_VAR

IF __ISVALIDREF(scConnector) THEN
	Main();
END_IF

ACTION Main:
{attribute 'conditionalshow'}
//Call parent function
SUPER^.Main();

//Call all functions
afb_ObjectInt_Out[1].tDataTimeOut := T#24H;
afb_ObjectInt_Out[1].eCommandType := _Domoticz_eCommandType.SwitchLight;
afb_ObjectInt_Out[1].eDataSource := _Domoticz_eDataSource.MQTT;
afb_ObjectInt_Out[1](scConnector := scConnector, 	uiIdentifier := uiIdentifier);

//Outputs
IF afb_ObjectInt_Out[1].xUpdateReceived THEN
	FOR wX := 1 TO 4 DO
		{warning disable C0196}
		//10 = 1 short, 20 = 1 long, 30 = 2 short, etc.
		axButtons_Short[wX] 	:= ((afb_ObjectInt_Out[1].iValueAct MOD ((wX*20) - 10)) = 0) AND (afb_ObjectInt_Out[1].iValueAct/((wX*20) - 10) = 1);
		axButtons_Long[wX] 	:= 	(afb_ObjectInt_Out[1].iValueAct MOD (wX*20)) = 0 AND (afb_ObjectInt_Out[1].iValueAct/(wX*20) = 1);
		{warning restore C0196}
	END_FOR
ELSE
	FOR wX := 1 TO 4 DO
		axButtons_Short[wX] 	:= FALSE;
		axButtons_Long[wX]		:= FALSE;
	END_FOR
END_IF 	

//Errors
fbEI_DataTimeOut.sInstanceName := sInstanceName;
fbEI_DataTimeOut.tErrorDelay := T#500MS;	//Give objects TIME TO be overruled BY other updates
fbEI_DataTimeOut(
	scConnector:= scConnector,
	xError:= xDataTimeOut_int
			AND (afb_ObjectInt_Out[1].xDataTimedOut),
	eErrorID:= Domoticz_eErrors.ObjectDataTimeOut
);
END_ACTION

END_FUNCTION_BLOCK
